FUNCTION_BLOCK FB_Director
VAR_INPUT
	//Panel Buttons
	Emergency :BOOL; //seta
	EndBatch  :BOOL;
	End		  :BOOL;
	Fail  	  :BOOL;
	Go        :BOOL; //marcha
	Manual 	  :BOOL; //manual
	Reboot 	  :BOOL;
	Restore   :BOOL;
	Stop      :BOOL; //parada

END_VAR
VAR_OUTPUT
	Mode : GEMMA := GEMMA.A6Inicializando;
	Pause : BOOL;
	Production : BOOL;
		
END_VAR
VAR
	ModeAns: GEMMA;
END_VAR

(* Define output commands*)
Pause := (Mode = A3ParadaEstado) 
		 OR (Mode = A4ParadaObtenida) 
		 OR (Mode = A5PreparandoTrasFallo)
		 OR (Mode = D1ParadaEmergencia) 
		 OR (Mode = D2TratamientoFallos);
Production := (Mode = A2ParaFinCiclo)
		   OR (Mode = A3ParadaEstado)
		   OR (Mode = F1ProduccionNormal)
		   OR (Mode = F2SecuenciaPreparacion)
		   OR (Mode = F3SecuenciaFinalizacion)
		   OR (Mode = F5VerificacionOrdenada)
		   OR (Mode = F6Probando)
		   OR (Mode = D3ProducirConFallos);
(* Choose mode *)

IF Reboot THEN
	Mode := A6Inicializando;
ELSIF Emergency THEN
	Mode := D1ParadaEmergencia;
END_IF

CASE Mode OF
	// ARRÈT 
	A1ParadaInicial:
	IF Manual THEN
		Mode := F4VerificacionSinOrden;
	ELSIF Go THEN
		Mode := F2SecuenciaPreparacion;
	END_IF
	
	A2ParaFinCiclo:
	IF Fail THEN
		ModeAns := A2ParaFinCiclo;
		Mode 	:= D2TratamientoFallos;
	ELSIF EndBatch THEN
		Mode := A1ParadaInicial;
	END_IF
	
	A5PreparandoTrasFallo: 
	IF Go THEN
		Mode := A1ParadaInicial;
	ELSIF Stop THEN
		Mode := A6Inicializando;
	END_IF
	
	A6Inicializando:
	IF Restore THEN
		Mode := A1ParadaInicial;
	ELSIF Manual THEN
		Mode := F4VerificacionSinOrden;
	END_IF
	
	// Fonctionnement
	F1ProduccionNormal: 
	IF Fail THEN
		ModeAns := A2ParaFinCiclo;
		Mode := D2TratamientoFallos;
	ELSIF EndBatch THEN
		Mode := F3SecuenciaFinalizacion;
	ELSIF Stop THEN
		Mode := A2ParaFinCiclo;
	END_IF
	
	F3SecuenciaFinalizacion: 
	IF End THEN
		Mode := A1ParadaInicial;
	END_IF
	
	F4VerificacionSinOrden:
	IF NOT Manual THEN
		Mode := A6Inicializando;
	ELSIF Fail THEN
		ModeAns := A2ParaFinCiclo;
		Mode := D2TratamientoFallos;
	END_IF
	
	// Défail
	D1ParadaEmergencia :
	IF NOT Emergency THEN
		Mode := A6Inicializando;
	END_IF
	
	D2TratamientoFallos:
	IF NOT Fail THEN
		Mode := A5PreparandoTrasFallo;
	END_IF
END_CASE

END_FUNCTION_BLOCK

(* stored: Version 1.1.0.1, ProductVersion 3.1.4024.6
   POU FB_Director: Id {6cbeff3c-1488-4cf2-8989-7affece50e4f}, SpecialFunc None *)
